FUNCTION MetricMaterialDimensions : BOOL
VAR_IN_OUT
	materials : ARRAY[*] OF Material;
END_VAR
VAR
	i : DINT;
END_VAR

FOR i:=LOWER_BOUND(materials, 1) TO UPPER_BOUND(materials, 1) BY 1 DO
	materials[i].lengthMM := TO_INT(materials[i].length * 25.4);
	materials[i].widthMM := TO_INT(materials[i].width * 25.4);
END_FOR

END_FUNCTION

(* stored: Version 1.1.0.1, ProductVersion 3.1.4024.11
   POU MetricMaterialDimensions: Id {c8d53307-fb53-44cd-9a7d-5bedc1c5b165}, SpecialFunc None *)
